TYPE T_CCS_CFG:
STRUCT
	site:     TrkSiteConstants;
END_STRUCT
END_TYPE

(* stored: Version 1.1.0.1, ProductVersion 3.1.4022.16
   DUT T_CCS_CFG: Id {560b22ba-8c55-4bb4-98cd-67316ecb02e0} *)
